# EPICS StreamDevice protocol: FW102/fw102.proto
# Communication protocol for FW102 Filter Wheel
# Oliver Copping
# 2023

Terminator = "\r"; # CR
InTemrinatorExtra = "> ";
OutTerminator = $Terminator;
InTerminator = $Terminator$InTemrinatorExtra; # CR + '> '

ReplyTimeout = 1000;
WriteTimeout = 1000;
ReadTimeout  = 1000;

getID       { out "*idn?"; in "*idn?\r%[ .a-zA-Z0-9]"; }

getPos      { out "pos?"; in "pos?\r%[0-9]"; }

setPos      { out "pos=%i"; }
